(* This function is for the Pirani MKS 317 connected to a 937A/B *)
(* This function block is used to provide protection and automatic turn on of ion gauges,
 it also manages the turn on of the AT_VAC boolean, and checks to make sure the pressure is good *)

FUNCTION_BLOCK FB_MKS317A
VAR_IN_OUT
	
END_VAR
VAR_INPUT
	
END_VAR
VAR_OUTPUT
	{attribute 'pytmc' := '
    pv: 
	'}
	PG : ST_VG;
END_VAR
VAR
	rV	:	REAL;
	rMinPressure: REAL := 1E-3;
	rDefaultVAC_SP: REAL :=5E-2; // Default 50 mT
	rValidLoBoundary	:	REAL := 0.2;//Manual page 61
	rValidHiBoundary	:	REAL := 9.7; //manual oage 61
	rDisconnectedBoundary	:	REAL := 0.17;
	rNoSensorBoundary	:	REAL := 10;
	(*IO*)
	i_iPRESS_R AT%I* :INT; // input Pressure // Link to analog Input
END_VAR

(* 937B Logarithmic Output Conversion *)
(* 5-20-2016, Alex Wallace and Scott Stubbs *)
(* 09-28-2018, Margaret Ghaly *)
(* This function will read the pressure from any gauge on a 937B. *)

rV := 10*INT_TO_REAL(PG.i_iPRESS_R)/32767;
PG.rPRESS := LREAL_TO_REAL(EXPT(10,((rV)/0.6)-12)); //manual page 61 937A


//Default setpoint 
IF PG.rVAC_SP = 0 THEN
	PG.rVAC_SP := rDefaultVAC_SP;
END_IF

IF (rV <=9.7 ) AND (rV>=0.6) THEN
	PG.eState := Valid; // normal
ELSIF rV >= 0.18 AND rV <= 0.22 THEN
	PG.eState := ValidLo; //LO
	PG.rPRESS := rMinPressure;
ELSIF rV > 9.7 AND rV<= 9.9 THEN
	PG.eState := ValidHi; //HIGH
ELSIF rV < 0.18 THEN
	PG.eState := GaugeDisconnected; //not on
	PG.rPRESS := -1;
ELSE
	PG.eState := PressInvalid; //other fault - could be no gauge, controller powering up etc
	PG.rPRESS := -1;
END_IF

(* Pressure OK check *)
(* Pressure gauge OK checks *)
PG.xPRESS_OK := (rV <=rValidHiBoundary ) AND (rV>=rDisconnectedBoundary);
//PG.xPRESS_OK := (PG.rPRESS >= rMinPressure);

(* Setpoint evaluation *)
PG.xAT_VAC := (*(PG.eState =Valid)*) PG.xPRESS_OK AND PG.rPRESS < PG.rVAC_SP;


(*soft io*)
IO();

ACTION IO:
PG.i_iPRESS_R :=i_iPRESS_R;
END_ACTION

END_FUNCTION_BLOCK

(* stored: Version 1.1.0.1, ProductVersion 3.1.4022.16
   POU FB_MKS317A: Id {5da6683a-653a-4dd9-bfe9-211b87873c21}, SpecialFunc None
   Action IO: Id {193cb751-e264-4d99-903a-eefc06eb5f23} *)
